TYPE HMIRFIDInterface :
STRUCT
	PermissionHardware	:	BOOL;
	PartPresent	:	BOOL;
	ExecuteCommand	:	BOOL;
	FMReading	:	BOOL;
	FMWritting	:	BOOL;
	ErrorActive	:	BOOL;
	SelectedCommand	:	WORD;
	ReadValue	:	WORD;
	WriteValue	:	WORD;
	SelectedMemoryIndex	:	WORD;
	StatusReader	:	WORD;
	CommandID	:	WORD;
	AllReadData	:	ARRAY[0..127] OF WORD;
	AllWriteData	:	ARRAY[0..127] OF WORD;
END_STRUCT
END_TYPE

(* stored: Version 1.1.0.1
   DUT HMIRFIDInterface: Id {1b526505-33bd-42a4-a645-94e60f72605b} *)
